TYPE U_UMC_Lenze_Status :

UNION
	Input: UINT;
	Data: T_UMC_Lenze_Status;
END_UNION

END_TYPE

(* stored: Version 1.1.0.1, ProductVersion 3.1.0.26
   DUT U_UMC_Lenze_Status: Id {e42cdc26-aacb-4ee9-a8e8-4ca5ab974d66} *)
